Staubli VAL3: readLogin.pgx

program readLogin(num x_nCamID (dimensions=1), string& x_sMsg[] (dimensions=1), bool& x_bError[] (dimensions=1))
  local num l_nChar
  local num l_nCount
begin
  //-----------------------------------------------------------------------
  //Header begin
  //Description of program
  // Read characters from socket until ":" is received
  //
  //Input parameters
  //  num x_nCamID :
  //    role : camera's ID
  //
  //Output parameters
  //  string x_sMsg:
  //    role : returns the error message
  //  bool x_bError :
  //    role : returns true if an error occurred and false otherwise
  //
  //Examples
  //  call readLogin(nCamID,"D5",l_nValue,x_bError)
  //
  //History
  //  Creation : 19-05-08 - f.Rob
  //Header end
  //-----------------------------------------------------------------------

  x_sMsg=""
  do
    l_nCount=sioGet(cCamera[x_nCamID].sSocket,l_nChar)
    //-1 : timeout for input communication has been reached
    if (l_nCount>-1) and (l_nChar>=32)
      x_sMsg=x_sMsg+chr(l_nChar)
    endIf
    x_bError=l_nCount<=-1
  until (chr(l_nChar)==":") or x_bError
  //Communication Error
  if x_bError
    cCamera[x_nCamID].nErrorCode=2
  endIf
  //Displays error message
  if bDebugProgram
    putln("ReadLogin : "+x_sMsg)
  endIf
end
